Staubli VAL3: selectedClear.pgx

program selectedClear()
begin
  if bSelectItem
    bSelectedItems[0] = true
    bSelectedItems[1] = true
    bSelectedItems[2] = true
    bSelectedItems[3] = true
    bSelectedItems[4] = true
    bSelectedItems[5] = true
  endIf
  bSelectItem  = false
  bSkipGlue[0] = false
end
